TYPE EL3152_HWTOPLC_PDOS :
	STRUCT
		
	
	Channel1 	AT %I* : EL3152_CHANNEL;
	Channel2 	AT %I* : EL3152_CHANNEL;



	END_STRUCT
END_TYPE

(* stored: Version 1.1.0.1, ProductVersion 3.1.4024.15
   DUT EL3152_HWTOPLC_PDOS: Id {d345304b-ec6e-4ea8-a50b-85857a128210} *)
